INTERFACE I_RpcServerConfig EXTENDS I_ServerConfig, I_RpcManagerConfig

END_INTERFACE

(* stored: Version 1.1.0.1, ProductVersion 3.1.4024.12
   Itf I_RpcServerConfig: Id {f1f1ac42-0ed5-4d02-93a4-3a3c64eacaab} *)
